(*
    Interpreter fixture. Exercises the Tc2_Standard WSTRING function set
    (WCONCAT, WDELETE, WFIND, WINSERT, WLEFT, WLEN, WMID, WREPLACE, WRIGHT)
    resolving through the native-function plugin/registry path
    (samples/xStunit.StandardStringPlugins), not a built-in intrinsic.

    Unlike CONCAT - an interpreter intrinsic, so a plugin counterpart would
    be unreachable - WCONCAT is NOT shadowed: the intrinsic is dispatched by
    exact ordinal name match on "CONCAT" (Engine.Expressions.cs), which
    "WCONCAT" does not hit, and no other intrinsic mentions it. It is
    therefore implemented as a plugin function here and covered below.

    WSTRING literals use "..." rather than STRING's '...'. Both are plain C#
    strings inside the interpreter, so the wide functions count UTF-16 code
    units - the same unit TwinCAT's WSTRING is defined in.
*)
FUNCTION_BLOCK FB_WideStringPluginTests EXTENDS TcUnit.FB_TestSuite

WLenReturnsTheCharacterCount();
WLenCountsWideCharactersNotBytes();
WLenOfEmptyIsZero();
WLeftReturnsTheLeftmostCharacters();
WLeftClampsWhenSizeExceedsLength();
WLeftReturnsEmptyForNonPositiveSize();
WRightReturnsTheRightmostCharacters();
WRightClampsWhenSizeExceedsLength();
WMidReturnsLenCharactersFromPos();
WMidClampsWhenPosPlusLenExceedsLength();
WMidReturnsEmptyWhenPosPastEnd();
WDeleteRemovesLenCharactersAtPos();
WDeleteClampsWhenPosPlusLenExceedsLength();
WInsertPlacesStr2AfterPos();
WInsertClampsPosBeyondEnd();
WReplaceSwapsCharactersForStr2();
WReplaceLeavesStringUnchangedWhenPosPastEnd();
WFindReturnsThePositionOfTheFirstMatch();
WFindReturnsZeroWhenNotFound();
WFindReturnsZeroForEmptyNeedle();
WConcatAppendsStr2ToStr1();
WConcatAppendsOptionalTrailingArgs();

METHOD PRIVATE WLenReturnsTheCharacterCount
VAR
	wsFullPath	: WSTRING(80) := "Root.Child.Leaf";
	nLength		: INT;
END_VAR
TEST('WLenReturnsTheCharacterCount');

nLength := WLEN(wsFullPath);

AssertEquals_INT(Expected := 15,
                  Actual := nLength,
                  Message := 'WLEN returns the wide-character count');

TEST_FINISHED();
END_METHOD

METHOD PRIVATE WLenCountsWideCharactersNotBytes
VAR
	wsAccented	: WSTRING(80) := "h$E9llo";
	nLength		: INT;
END_VAR
TEST('WLenCountsWideCharactersNotBytes');

(* $E9 is a single non-ASCII wide character; WLEN counts characters, not
   the bytes a narrow encoding would need for it. *)
nLength := WLEN(wsAccented);

AssertEquals_INT(Expected := 5,
                  Actual := nLength,
                  Message := 'WLEN counts wide characters, not encoded bytes');

TEST_FINISHED();
END_METHOD

METHOD PRIVATE WLenOfEmptyIsZero
VAR
	nLength		: INT;
END_VAR
TEST('WLenOfEmptyIsZero');

nLength := WLEN("");

AssertEquals_INT(Expected := 0,
                  Actual := nLength,
                  Message := 'WLEN of an empty WSTRING is 0');

TEST_FINISHED();
END_METHOD

METHOD PRIVATE WLeftReturnsTheLeftmostCharacters
VAR
	wsFullPath	: WSTRING(80) := "Root.Child.Leaf.Extra";
	nIndex		: INT := 16;
	wsResult	: WSTRING(80);
END_VAR
TEST('WLeftReturnsTheLeftmostCharacters');

wsResult := WLEFT(wsFullPath, nIndex - 1);

AssertEquals_WSTRING(Expected := "Root.Child.Leaf",
                      Actual := wsResult,
                      Message := 'WLEFT returns the leftmost SIZE characters');

TEST_FINISHED();
END_METHOD

METHOD PRIVATE WLeftClampsWhenSizeExceedsLength
VAR
	wsResult	: WSTRING(80);
END_VAR
TEST('WLeftClampsWhenSizeExceedsLength');

wsResult := WLEFT("abc", 10);

AssertEquals_WSTRING(Expected := "abc",
                      Actual := wsResult,
                      Message := 'WLEFT clamps SIZE to the length of STR');

TEST_FINISHED();
END_METHOD

METHOD PRIVATE WLeftReturnsEmptyForNonPositiveSize
VAR
	wsResult	: WSTRING(80);
END_VAR
TEST('WLeftReturnsEmptyForNonPositiveSize');

wsResult := WLEFT("abc", -4);

AssertEquals_WSTRING(Expected := "",
                      Actual := wsResult,
                      Message := 'WLEFT clamps a negative SIZE to 0');

TEST_FINISHED();
END_METHOD

METHOD PRIVATE WRightReturnsTheRightmostCharacters
VAR
	wsFullPath	: WSTRING(80) := "Root.Child.Leaf";
	nPos		: INT := 5;
	wsResult	: WSTRING(80);
END_VAR
TEST('WRightReturnsTheRightmostCharacters');

wsResult := WRIGHT(wsFullPath, WLEN(wsFullPath) - nPos);

AssertEquals_WSTRING(Expected := "Child.Leaf",
                      Actual := wsResult,
                      Message := 'WRIGHT returns the rightmost SIZE characters');

TEST_FINISHED();
END_METHOD

METHOD PRIVATE WRightClampsWhenSizeExceedsLength
VAR
	wsResult	: WSTRING(80);
END_VAR
TEST('WRightClampsWhenSizeExceedsLength');

wsResult := WRIGHT("abc", 10);

AssertEquals_WSTRING(Expected := "abc",
                      Actual := wsResult,
                      Message := 'WRIGHT clamps SIZE to the length of STR');

TEST_FINISHED();
END_METHOD

METHOD PRIVATE WMidReturnsLenCharactersFromPos
VAR
	wsFullPath	: WSTRING(80) := "Root.Child.Leaf";
	nLen		: INT := 5;
	nPos		: INT := 6;
	wsResult	: WSTRING(80);
END_VAR
TEST('WMidReturnsLenCharactersFromPos');

wsResult := WMID(wsFullPath, nLen, nPos);

AssertEquals_WSTRING(Expected := "Child",
                      Actual := wsResult,
                      Message := 'WMID returns LEN characters starting at POS');

TEST_FINISHED();
END_METHOD

METHOD PRIVATE WMidClampsWhenPosPlusLenExceedsLength
VAR
	wsResult	: WSTRING(80);
END_VAR
TEST('WMidClampsWhenPosPlusLenExceedsLength');

(* POS=3, LEN=100 asks for far more than remains of a 5-character string. *)
wsResult := WMID("abcde", 100, 3);

AssertEquals_WSTRING(Expected := "cde",
                      Actual := wsResult,
                      Message := 'WMID clamps LEN to what remains from POS');

TEST_FINISHED();
END_METHOD

METHOD PRIVATE WMidReturnsEmptyWhenPosPastEnd
VAR
	wsResult	: WSTRING(80);
END_VAR
TEST('WMidReturnsEmptyWhenPosPastEnd');

wsResult := WMID("abcde", 2, 99);

AssertEquals_WSTRING(Expected := "",
                      Actual := wsResult,
                      Message := 'WMID returns an empty WSTRING when POS is past the end');

TEST_FINISHED();
END_METHOD

METHOD PRIVATE WDeleteRemovesLenCharactersAtPos
VAR
	wsFullPath	: WSTRING(80) := "Root.Child]";
	nPos		: INT := 11;
	wsResult	: WSTRING(80);
END_VAR
TEST('WDeleteRemovesLenCharactersAtPos');

wsResult := WDELETE(wsFullPath, 1, nPos);

AssertEquals_WSTRING(Expected := "Root.Child",
                      Actual := wsResult,
                      Message := 'WDELETE removes LEN characters at POS');

TEST_FINISHED();
END_METHOD

METHOD PRIVATE WDeleteClampsWhenPosPlusLenExceedsLength
VAR
	wsResult	: WSTRING(80);
END_VAR
TEST('WDeleteClampsWhenPosPlusLenExceedsLength');

(* POS=3, LEN=100 asks to remove past the end of a 5-character string. *)
wsResult := WDELETE("abcde", 100, 3);

AssertEquals_WSTRING(Expected := "ab",
                      Actual := wsResult,
                      Message := 'WDELETE clamps LEN to the remaining length');

TEST_FINISHED();
END_METHOD

METHOD PRIVATE WInsertPlacesStr2AfterPos
VAR
	wsBase		: WSTRING(80) := "Root.Leaf";
	wsInsert	: WSTRING(80) := "Child.";
	nPos		: INT := 5;
	wsResult	: WSTRING(80);
END_VAR
TEST('WInsertPlacesStr2AfterPos');

wsResult := WINSERT(wsBase, wsInsert, nPos);

AssertEquals_WSTRING(Expected := "Root.Child.Leaf",
                      Actual := wsResult,
                      Message := 'WINSERT places STR2 immediately after POS');

TEST_FINISHED();
END_METHOD

METHOD PRIVATE WInsertClampsPosBeyondEnd
VAR
	wsResult	: WSTRING(80);
END_VAR
TEST('WInsertClampsPosBeyondEnd');

wsResult := WINSERT("abc", "XY", 99);

AssertEquals_WSTRING(Expected := "abcXY",
                      Actual := wsResult,
                      Message := 'WINSERT clamps POS to the end of STR1');

TEST_FINISHED();
END_METHOD

METHOD PRIVATE WReplaceSwapsCharactersForStr2
VAR
	wsFullPath	: WSTRING(80) := "Root[0].Leaf";
	nPos		: INT := 5;
	wsResult	: WSTRING(80);
END_VAR
TEST('WReplaceSwapsCharactersForStr2');

wsResult := WREPLACE(wsFullPath, "_", 1, nPos);

AssertEquals_WSTRING(Expected := "Root_0].Leaf",
                      Actual := wsResult,
                      Message := 'WREPLACE swaps L characters at P for STR2');

TEST_FINISHED();
END_METHOD

METHOD PRIVATE WReplaceLeavesStringUnchangedWhenPosPastEnd
VAR
	wsResult	: WSTRING(80);
END_VAR
TEST('WReplaceLeavesStringUnchangedWhenPosPastEnd');

wsResult := WREPLACE("abcde", "XY", 2, 99);

AssertEquals_WSTRING(Expected := "abcde",
                      Actual := wsResult,
                      Message := 'WREPLACE is a no-op when P is past the end of STR1');

TEST_FINISHED();
END_METHOD

METHOD PRIVATE WFindReturnsThePositionOfTheFirstMatch
VAR
	wsFullPath	: WSTRING(80) := "Root.Child.Leaf";
	nSeparator	: INT;
END_VAR
TEST('WFindReturnsThePositionOfTheFirstMatch');

nSeparator := WFIND(wsFullPath, ".");

AssertEquals_INT(Expected := 5,
                  Actual := nSeparator,
                  Message := 'WFIND returns the 1-based position of the first match');

TEST_FINISHED();
END_METHOD

METHOD PRIVATE WFindReturnsZeroWhenNotFound
VAR
	nResult		: INT;
END_VAR
TEST('WFindReturnsZeroWhenNotFound');

nResult := WFIND("abcde", "z");

AssertEquals_INT(Expected := 0,
                  Actual := nResult,
                  Message := 'WFIND returns 0 when STR2 is not found');

TEST_FINISHED();
END_METHOD

METHOD PRIVATE WFindReturnsZeroForEmptyNeedle
VAR
	nResult		: INT;
END_VAR
TEST('WFindReturnsZeroForEmptyNeedle');

nResult := WFIND("abcde", "");

AssertEquals_INT(Expected := 0,
                  Actual := nResult,
                  Message := 'WFIND returns 0 for an empty STR2');

TEST_FINISHED();
END_METHOD

METHOD PRIVATE WConcatAppendsStr2ToStr1
VAR
	wsLeft		: WSTRING(80) := "Root.";
	wsResult	: WSTRING(80);
END_VAR
TEST('WConcatAppendsStr2ToStr1');

(* Unlike CONCAT (an interpreter intrinsic), WCONCAT is
   not intercepted before native-function dispatch - the intrinsic matches
   the method name "CONCAT" exactly - so this call reaches the plugin. *)
wsResult := WCONCAT(wsLeft, "Leaf");

AssertEquals_WSTRING(Expected := "Root.Leaf",
                      Actual := wsResult,
                      Message := 'WCONCAT appends STR2 to STR1');

TEST_FINISHED();
END_METHOD

METHOD PRIVATE WConcatAppendsOptionalTrailingArgs
VAR
	wsResult	: WSTRING(80);
END_VAR
TEST('WConcatAppendsOptionalTrailingArgs');

(* STR3..STR10 are optional trailing arguments, same shape as the CONCAT
   intrinsic (Engine.Expressions.cs's ConcatParamNames). *)
wsResult := WCONCAT("a", "b", "c", "d");

AssertEquals_WSTRING(Expected := "abcd",
                      Actual := wsResult,
                      Message := 'WCONCAT appends every supplied STRn in declared order');

TEST_FINISHED();
END_METHOD

END_FUNCTION_BLOCK

(* stored: Version 1.1.0.1, ProductVersion 3.1.4026.18
   POU FB_WideStringPluginTests: Id {93190000-0000-4a1a-8b1b-000000000000}, SpecialFunc None
   Method WLenReturnsTheCharacterCount: Id {93190000-0000-4a1a-8b1b-000000000001}
   Method WLenCountsWideCharactersNotBytes: Id {93190000-0000-4a1a-8b1b-000000000002}
   Method WLenOfEmptyIsZero: Id {93190000-0000-4a1a-8b1b-000000000003}
   Method WLeftReturnsTheLeftmostCharacters: Id {93190000-0000-4a1a-8b1b-000000000004}
   Method WLeftClampsWhenSizeExceedsLength: Id {93190000-0000-4a1a-8b1b-000000000005}
   Method WLeftReturnsEmptyForNonPositiveSize: Id {93190000-0000-4a1a-8b1b-000000000006}
   Method WRightReturnsTheRightmostCharacters: Id {93190000-0000-4a1a-8b1b-000000000007}
   Method WRightClampsWhenSizeExceedsLength: Id {93190000-0000-4a1a-8b1b-000000000008}
   Method WMidReturnsLenCharactersFromPos: Id {93190000-0000-4a1a-8b1b-000000000009}
   Method WMidClampsWhenPosPlusLenExceedsLength: Id {93190000-0000-4a1a-8b1b-00000000000a}
   Method WMidReturnsEmptyWhenPosPastEnd: Id {93190000-0000-4a1a-8b1b-00000000000b}
   Method WDeleteRemovesLenCharactersAtPos: Id {93190000-0000-4a1a-8b1b-00000000000c}
   Method WDeleteClampsWhenPosPlusLenExceedsLength: Id {93190000-0000-4a1a-8b1b-00000000000d}
   Method WInsertPlacesStr2AfterPos: Id {93190000-0000-4a1a-8b1b-00000000000e}
   Method WInsertClampsPosBeyondEnd: Id {93190000-0000-4a1a-8b1b-00000000000f}
   Method WReplaceSwapsCharactersForStr2: Id {93190000-0000-4a1a-8b1b-000000000010}
   Method WReplaceLeavesStringUnchangedWhenPosPastEnd: Id {93190000-0000-4a1a-8b1b-000000000011}
   Method WFindReturnsThePositionOfTheFirstMatch: Id {93190000-0000-4a1a-8b1b-000000000012}
   Method WFindReturnsZeroWhenNotFound: Id {93190000-0000-4a1a-8b1b-000000000013}
   Method WFindReturnsZeroForEmptyNeedle: Id {93190000-0000-4a1a-8b1b-000000000014}
   Method WConcatAppendsStr2ToStr1: Id {93190000-0000-4a1a-8b1b-000000000015}
   Method WConcatAppendsOptionalTrailingArgs: Id {93190000-0000-4a1a-8b1b-000000000016} *)
